LIN {X 0,Y 81.838,Z 446.637,A -85,B 0,C 180,E1 -31138.318,E2 -31138.318} C_VEL
LIN {X 0,Y 84.588,Z 433.507,A -85,B 0,C 180,E1 -31138.672,E2 -31138.672} C_VEL
LIN {X 0,Y 85.989,Z 422.643,A -85,B 0,C 180,E1 -31138.95,E2 -31138.95} C_VEL
LIN {X 0,Y 85.565,Z 419.537,A -85,B 0,C 180,E1 -31144.015,E2 -31144.015} C_VEL
LIN {X 0,Y 85.47,Z 419.121,A -85,B 0,C 180,E1 -31146.346,E2 -31146.346} C_VEL
LIN {X 0,Y 85.574,Z 420.483,A -85,B 0,C 180,E1 -31152.716,E2 -31152.716} C_VEL
LIN {X 0,Y 85.929,Z 422.6,A -85,B 0,C 180,E1 -31156.35,E2 -31156.35} C_VEL
LIN {X 0,Y 84.135,Z 435.518,A -85,B 0,C 180,E1 -31156.663,E2 -31156.663} C_VEL
LIN {X 0,Y 80.891,Z 449.175,A -85,B 0,C 180,E1 -31157.094,E2 -31157.094} C_VEL
LIN {X 0,Y 76.93,Z 460.689,A -85,B 0,C 180,E1 -31157.829,E2 -31157.829} C_VEL
LIN {X 0,Y 71.448,Z 472.538,A -85,B 0,C 180,E1 -31158.755,E2 -31158.755} C_VEL
LIN {X 0,Y 65.417,Z 482.814,A -85,B 0,C 180,E1 -31159.917,E2 -31159.917} C_VEL
LIN {X 0,Y 59.027,Z 491.818,A -85,B 0,C 180,E1 -31161.492,E2 -31161.492} C_VEL
LIN {X 0,Y 50.481,Z 501.765,A -85,B 0,C 180,E1 -31164.204,E2 -31164.204} C_VEL
LIN {X 0,Y 41.76,Z 510.143,A -85,B 0,C 180,E1 -31167.896,E2 -31167.896} C_VEL
LIN {X 0,Y 36.402,Z 514.585,A -85,B 0,C 180,E1 -31170.912,E2 -31170.912} C_VEL
LIN {X 0,Y 31.72,Z 517.965,A -85,B 0,C 180,E1 -31173.277,E2 -31173.277} C_VEL
LIN {X 0,Y 23.201,Z 522.944,A -85,B 0,C 180,E1 -31175.169,E2 -31175.169} C_VEL
LIN {X 0,Y 16.084,Z 526.477,A -85,B 0,C 180,E1 -31177.474,E2 -31177.474} C_VEL
LIN {X 0,Y 10.911,Z 528.904,A -85,B 0,C 180,E1 -31184.743,E2 -31184.743} C_VEL
LIN {X 0,Y 9.359,Z 529.652,A -85,B 0,C 180,E1 -31190.249,E2 -31190.249} C_VEL
LIN {X 0,Y 5.866,Z 533.194,A -85,B 0,C 180,E1 -31266.672,E2 -31266.672} C_VEL
LIN {X 0,Y 14.149,Z 536.113,A -85,B 0,C 180,E1 -31313.053,E2 -31313.053} C_VEL
LIN {X 0,Y 21.077,Z 537.497,A -85,B 0,C 180,E1 -31321.144,E2 -31321.144} C_VEL
LIN {X 0,Y 28.229,Z 538.473,A -85,B 0,C 180,E1 -31325.459,E2 -31325.459} C_VEL
LIN {X 0,Y 28.277,Z 538.497,A -85,B 0,C 180,E1 -31326.4,E2 -31326.4} C_VEL
LIN {X 0,Y 14.86,Z 536.532,A -85,B 0,C 180,E1 -31339.064,E2 -31339.064} C_VEL
LIN {X 0,Y 6.839,Z 534.003,A -85,B 0,C 180,E1 -31379.184,E2 -31379.184} C_VEL
LIN {X 0,Y 6.067,Z 532.96,A -85,B 0,C 180,E1 -31410.099,E2 -31410.099} C_VEL
LIN {X 0,Y 11.691,Z 528.915,A -85,B 0,C 180,E1 -31474.506,E2 -31474.506} C_VEL
LIN {X 0,Y 23.106,Z 522.633,A -85,B 0,C 180,E1 -31491.486,E2 -31491.486} C_VEL
LIN {X 0,Y 33.453,Z 515.774,A -85,B 0,C 180,E1 -31496.564,E2 -31496.564} C_VEL
LIN {X 0,Y 42.181,Z 508.715,A -85,B 0,C 180,E1 -31499.341,E2 -31499.341} C_VEL
LIN {X 0,Y 50.965,Z 500.289,A -85,B 0,C 180,E1 -31500.521,E2 -31500.521} C_VEL
LIN {X 0,Y 58.891,Z 490.996,A -85,B 0,C 180,E1 -31501.575,E2 -31501.575} C_VEL
LIN {X 0,Y 64.188,Z 483.557,A -85,B 0,C 180,E1 -31502.219,E2 -31502.219} C_VEL
LIN {X 0,Y 71.246,Z 471.606,A -85,B 0,C 180,E1 -31502.685,E2 -31502.685} C_VEL
LIN {X 0,Y 76.986,Z 458.755,A -85,B 0,C 180,E1 -31503.031,E2 -31503.031} C_VEL
LIN {X 0,Y 81.207,Z 445.716,A -85,B 0,C 180,E1 -31503.307,E2 -31503.307} C_VEL
LIN {X 0,Y 83.825,Z 433.16,A -85,B 0,C 180,E1 -31503.469,E2 -31503.469} C_VEL
LIN {X 0,Y 84.631,Z 427.284,A -85,B 0,C 180,E1 -31503.645,E2 -31503.645} C_VEL
LIN {X 0,Y 84.615,Z 426.627,A -85,B 0,C 180,E1 -31504.763,E2 -31504.763} C_VEL
LIN {X 0,Y 84.581,Z 427.089,A -85,B 0,C 180,E1 -31511.077,E2 -31511.077} C_VEL
LIN {X 0,Y 84.594,Z 427.411,A -85,B 0,C 180,E1 -31511.695,E2 -31511.695} C_VEL
LIN {X 0,Y 82.44,Z 440.278,A -85,B 0,C 180,E1 -31511.882,E2 -31511.882} C_VEL
LIN {X 0,Y 78.624,Z 453.875,A -85,B 0,C 180,E1 -31512.237,E2 -31512.237} C_VEL
LIN {X 0,Y 73.685,Z 466.314,A -85,B 0,C 180,E1 -31512.797,E2 -31512.797} C_VEL
LIN {X 0,Y 67.706,Z 477.645,A -85,B 0,C 180,E1 -31513.272,E2 -31513.272} C_VEL
LIN {X 0,Y 60.758,Z 488.161,A -85,B 0,C 180,E1 -31514.325,E2 -31514.325} C_VEL
LIN {X 0,Y 52.81,Z 497.928,A -85,B 0,C 180,E1 -31515.545,E2 -31515.545} C_VEL
LIN {X 0,Y 44.162,Z 506.66,A -85,B 0,C 180,E1 -31517.238,E2 -31517.238} C_VEL
LIN {X 0,Y 33.699,Z 515.241,A -85,B 0,C 180,E1 -31520.153,E2 -31520.153} C_VEL
LIN {X 0,Y 23.372,Z 522.119,A -85,B 0,C 180,E1 -31525.503,E2 -31525.503} C_VEL
LIN {X 0,Y 13.372,Z 527.633,A -85,B 0,C 180,E1 -31537.893,E2 -31537.893} C_VEL
LIN {X 0,Y 9.359,Z 529.652,A -85,B 0,C 180,E1 -31550.249,E2 -31550.249} C_VEL
LIN {X 0,Y 8.403,Z 531.503,A -85,B 0,C 180,E1 -31555.375,E2 -31555.375} C_VEL
LIN {X 0,Y 8.403,Z 600,A -85,B 0,C 180,E1 -31555.375,E2 -31555.375} C_VEL
LIN {X 0,Y 8.403,Z 600,A -85,B 0,C 180,E1 -31555.375,E2 -31555.375}

QRS_NEXT_CUT()

QRS_NEXT()
QRS_HOME()

END
